{attribute 'linkalways'} 
{attribute 'no_explicit_call' := 'This FB is a CLASS and must be accessed using methods or properties'}
{attribute 'enable_dynamic_creation'}
FUNCTION_BLOCK Node_F_VN_FillContainer_TcVnVector2_DINT EXTENDS VisionNode
VAR
    ipContainer : _ITcVnContainer;
    aValue : _TcVnVector2_DINT;
    hrPrev : _HRESULT(S_OK);
    hresult : _HRESULT(S_OK);
END_VAR

METHOD PUBLIC  Clone : I_Node
VAR
    pNode : POINTER TO Node_F_VN_FillContainer_TcVnVector2_DINT;
END_VAR
pNode := __NEW(Node_F_VN_FillContainer_TcVnVector2_DINT);
Clone := pNode^;
END_METHOD

METHOD FB_init : BOOL
VAR_INPUT
    bInitRetains : BOOL; // if TRUE, the retain variables are initialized (warm start / cold start)
    bInCopyCode : BOOL;  // if TRUE, the instance afterwards gets moved into the copy code (online change)
END_VAR
AddInput('ipContainer', ipContainer);
AddInput('aValue', aValue);
AddInput('hrPrev', hrPrev);
AddOutput('ipContainer', ipContainer);
AddOutput('hresult',hresult);
END_METHOD

METHOD PROTECTED OnExecute : HRESULT
hresult.Value := F_VN_FillContainer_TcVnVector2_DINT(
    ipContainer := ipContainer.Value,
    aValue := aValue.Value,
    hrPrev:= hrPrev.Value);
END_METHOD

METHOD PUBLIC PreExecutionCheck
VAR_INPUT
    Check : I_PreExecutionChecks;
END_VAR
Check.IsTrue(ipContainer.IsValid, 'ipContainer must be a valid container');
END_METHOD

END_FUNCTION_BLOCK

(* stored: Version 1.1.0.1, ProductVersion 3.1.4024.13
   POU Node_F_VN_FillContainer_TcVnVector2_DINT: Id {f3990d17-1a9a-49b9-afb4-68bc099868a5}, SpecialFunc None
   Folder Constructor: Id {6644ef2f-12cf-4833-b2f2-79e6c63d3984}
   Method Clone: Id {edc67da6-78ee-4607-8933-b26462f1adbd}
   Method FB_init: Id {11bcbd4f-457b-4563-a1cd-967f2b13f037}
   Method OnExecute: Id {d08781a8-da18-4bdc-b1bf-04f4a7e2cecf}
   Method PreExecutionCheck: Id {223a612c-bd7f-4c0a-9147-8928b1dae0d8} *)
